// TwinCAT 3 PLC project PLC_PROJ
// ProgramVersion: 3.1.4026.15
// libraries:
//   Tc2_EtherCAT, * (Beckhoff Automation GmbH)
//   Tc2_IoFunctions, * (Beckhoff Automation GmbH)
//   Tc2_SerialCom, * (Beckhoff Automation GmbH)
//   Tc2_Standard, * (Beckhoff Automation GmbH)
//   Tc2_System, * (Beckhoff Automation GmbH)
// project tree:
//   DUTs/ CAN_IFACE_QUEUE.TcDUT, CAN_MSG.TcDUT, CAN_MsgSlot.TcDUT
//   GVLs/ ANALOG.TcGVL, EL6751_GVLs.TcGVL, GLOBAL_VARS.TcGVL
//   / PlcTask.TcTTO
//   POUs/CanHelpers/ F_ComposeSlot.TcPOU, F_ParseSlot.TcPOU
//   POUs/ MAIN.TcPOU
//   POUs/PsuHelpers/ BytesToUInt16.TcPOU, CurrentToRaw.TcPOU, RawToCurrent.TcPOU, RawToVoltage.TcPOU, VoltageToRaw.TcPOU
//   POUs/PsuIface/ FB_PowerSupply.TcPOU
// real-time tasks:
//   TASK PlcTask: cycle T#100000us, priority 20, ADS port 350
// I/O:
//   DEVICE Device 1 (EtherCAT), AmsNetId 5.156.240.208.2.1
//     Term 1 (EK1200) [EK1200-7000 EtherCAT Power supply (1,5A E-Bus)]
//       Term 2 (EL2008) [EL2008 8Ch. Dig. Output 24V, 0.5A]
//       Term 3 (EL3174-0042) [EL3174-0042 4Ch. Ana. Input +/-30V, +/-60V 16 Bit, Isolated Channels]
//       Term 4 (EL3692) [EL3692 2Ch. resistance measurement terminal]
//       Term 5 (EL6751) [EL6751 CANopen Master]
//       Term 6 (EL6631) [EL6631 PROFINET IO Controller]
//       Term 7 (EL9011) [EL9011 End Terminal]
//   DEVICE Device 2 (NOV-DP-RAM)
//   DEVICE Device 3 (Onboard I/O Device), AmsNetId 5.156.240.208.4.1
//     Term 1 (CX7028) [CX7028-0000-0121]
//       modules: Module 1 (DIO_2x), Module 2 (Empty Module), Module 3 (DIO_2x), Module 4 (Empty Module), Module 5 (DI_2x), Module 6 (Empty Module), Module 7 (DI_2x), Module 8 (Empty Module)
//   DEVICE Device 4 (COM Port)
//   DEVICE Device 5 (COM Port)
//   DEVICE Device 6 (EL6751), AmsNetId 5.156.240.208.7.1
//     Box 9 (CAN Interface)
// variable links:
//   PLC_PROJ/PLC_PROJ Instance <-> Device 1 (EtherCAT)/Term 1 (EK1200)/Term 2 (EL2008)
//     PlcTask Outputs/GLOBAL_VARS.DO_EL2008_OUT_2 <-> Channel 2/Output
//     PlcTask Outputs/GLOBAL_VARS.DO_EL2008_OUT_4 <-> Channel 4/Output
//     PlcTask Outputs/GLOBAL_VARS.DO_EL2008_OUT_5 <-> Channel 5/Output
//     PlcTask Outputs/GLOBAL_VARS.DO_EL2008_OUT_6 <-> Channel 6/Output
//     PlcTask Outputs/GLOBAL_VARS.DO_EL2008_OUT_7 <-> Channel 7/Output
//     PlcTask Outputs/GLOBAL_VARS.DO_EL2008_OUT_8 <-> Channel 8/Output
//     PlcTask Outputs/GLOBAL_VARS.DO_EL2008_RELAY_0 <-> Channel 1/Output
//     PlcTask Outputs/GLOBAL_VARS.DO_EL2008_RELAY_1 <-> Channel 3/Output
//   PLC_PROJ/PLC_PROJ Instance <-> Device 4 (COM Port)
//     PlcTask Inputs/GLOBAL_VARS.X003_In/D[0] <-> Inputs/Data1
//     PlcTask Inputs/GLOBAL_VARS.X003_In/D[10] <-> Inputs/Data11
//     PlcTask Inputs/GLOBAL_VARS.X003_In/D[11] <-> Inputs/Data12
//     PlcTask Inputs/GLOBAL_VARS.X003_In/D[12] <-> Inputs/Data13
//     PlcTask Inputs/GLOBAL_VARS.X003_In/D[13] <-> Inputs/Data14
//     PlcTask Inputs/GLOBAL_VARS.X003_In/D[14] <-> Inputs/Data15
//     PlcTask Inputs/GLOBAL_VARS.X003_In/D[15] <-> Inputs/Data16
//     PlcTask Inputs/GLOBAL_VARS.X003_In/D[16] <-> Inputs/Data17
//     PlcTask Inputs/GLOBAL_VARS.X003_In/D[17] <-> Inputs/Data18
//     PlcTask Inputs/GLOBAL_VARS.X003_In/D[18] <-> Inputs/Data19
//     PlcTask Inputs/GLOBAL_VARS.X003_In/D[19] <-> Inputs/Data20
//     PlcTask Inputs/GLOBAL_VARS.X003_In/D[1] <-> Inputs/Data2
//     PlcTask Inputs/GLOBAL_VARS.X003_In/D[20] <-> Inputs/Data21
//     PlcTask Inputs/GLOBAL_VARS.X003_In/D[21] <-> Inputs/Data22
//     PlcTask Inputs/GLOBAL_VARS.X003_In/D[22] <-> Inputs/Data23
//     PlcTask Inputs/GLOBAL_VARS.X003_In/D[23] <-> Inputs/Data24
//     PlcTask Inputs/GLOBAL_VARS.X003_In/D[24] <-> Inputs/Data25
//     PlcTask Inputs/GLOBAL_VARS.X003_In/D[25] <-> Inputs/Data26
//     PlcTask Inputs/GLOBAL_VARS.X003_In/D[26] <-> Inputs/Data27
//     PlcTask Inputs/GLOBAL_VARS.X003_In/D[27] <-> Inputs/Data28
//     PlcTask Inputs/GLOBAL_VARS.X003_In/D[28] <-> Inputs/Data29
//     PlcTask Inputs/GLOBAL_VARS.X003_In/D[29] <-> Inputs/Data30
//     PlcTask Inputs/GLOBAL_VARS.X003_In/D[2] <-> Inputs/Data3
//     PlcTask Inputs/GLOBAL_VARS.X003_In/D[30] <-> Inputs/Data31
//     PlcTask Inputs/GLOBAL_VARS.X003_In/D[31] <-> Inputs/Data32
//     PlcTask Inputs/GLOBAL_VARS.X003_In/D[32] <-> Inputs/Data33
//     PlcTask Inputs/GLOBAL_VARS.X003_In/D[33] <-> Inputs/Data34
//     PlcTask Inputs/GLOBAL_VARS.X003_In/D[34] <-> Inputs/Data35
//     PlcTask Inputs/GLOBAL_VARS.X003_In/D[35] <-> Inputs/Data36
//     PlcTask Inputs/GLOBAL_VARS.X003_In/D[36] <-> Inputs/Data37
//     PlcTask Inputs/GLOBAL_VARS.X003_In/D[37] <-> Inputs/Data38
//     PlcTask Inputs/GLOBAL_VARS.X003_In/D[38] <-> Inputs/Data39
//     PlcTask Inputs/GLOBAL_VARS.X003_In/D[39] <-> Inputs/Data40
//     PlcTask Inputs/GLOBAL_VARS.X003_In/D[3] <-> Inputs/Data4
//     PlcTask Inputs/GLOBAL_VARS.X003_In/D[40] <-> Inputs/Data41
//     PlcTask Inputs/GLOBAL_VARS.X003_In/D[41] <-> Inputs/Data42
//     PlcTask Inputs/GLOBAL_VARS.X003_In/D[42] <-> Inputs/Data43
//     PlcTask Inputs/GLOBAL_VARS.X003_In/D[43] <-> Inputs/Data44
//     PlcTask Inputs/GLOBAL_VARS.X003_In/D[44] <-> Inputs/Data45
//     PlcTask Inputs/GLOBAL_VARS.X003_In/D[45] <-> Inputs/Data46
//     PlcTask Inputs/GLOBAL_VARS.X003_In/D[46] <-> Inputs/Data47
//     PlcTask Inputs/GLOBAL_VARS.X003_In/D[47] <-> Inputs/Data48
//     PlcTask Inputs/GLOBAL_VARS.X003_In/D[48] <-> Inputs/Data49
//     PlcTask Inputs/GLOBAL_VARS.X003_In/D[49] <-> Inputs/Data50
//     PlcTask Inputs/GLOBAL_VARS.X003_In/D[4] <-> Inputs/Data5
//     PlcTask Inputs/GLOBAL_VARS.X003_In/D[50] <-> Inputs/Data51
//     PlcTask Inputs/GLOBAL_VARS.X003_In/D[51] <-> Inputs/Data52
//     PlcTask Inputs/GLOBAL_VARS.X003_In/D[52] <-> Inputs/Data53
//     PlcTask Inputs/GLOBAL_VARS.X003_In/D[53] <-> Inputs/Data54
//     PlcTask Inputs/GLOBAL_VARS.X003_In/D[54] <-> Inputs/Data55
//     PlcTask Inputs/GLOBAL_VARS.X003_In/D[55] <-> Inputs/Data56
//     PlcTask Inputs/GLOBAL_VARS.X003_In/D[56] <-> Inputs/Data57
//     PlcTask Inputs/GLOBAL_VARS.X003_In/D[57] <-> Inputs/Data58
//     PlcTask Inputs/GLOBAL_VARS.X003_In/D[58] <-> Inputs/Data59
//     PlcTask Inputs/GLOBAL_VARS.X003_In/D[59] <-> Inputs/Data60
//     PlcTask Inputs/GLOBAL_VARS.X003_In/D[5] <-> Inputs/Data6
//     PlcTask Inputs/GLOBAL_VARS.X003_In/D[60] <-> Inputs/Data61
//     PlcTask Inputs/GLOBAL_VARS.X003_In/D[61] <-> Inputs/Data62
//     PlcTask Inputs/GLOBAL_VARS.X003_In/D[62] <-> Inputs/Data63
//     PlcTask Inputs/GLOBAL_VARS.X003_In/D[63] <-> Inputs/Data64
//     PlcTask Inputs/GLOBAL_VARS.X003_In/D[6] <-> Inputs/Data7
//     PlcTask Inputs/GLOBAL_VARS.X003_In/D[7] <-> Inputs/Data8
//     PlcTask Inputs/GLOBAL_VARS.X003_In/D[8] <-> Inputs/Data9
//     PlcTask Inputs/GLOBAL_VARS.X003_In/D[9] <-> Inputs/Data10
//     PlcTask Inputs/GLOBAL_VARS.X003_In/SerStatus <-> Inputs/Status
//     PlcTask Outputs/GLOBAL_VARS.X003_Out/D[0] <-> Outputs/Data1
//     PlcTask Outputs/GLOBAL_VARS.X003_Out/D[10] <-> Outputs/Data11
//     PlcTask Outputs/GLOBAL_VARS.X003_Out/D[11] <-> Outputs/Data12
//     PlcTask Outputs/GLOBAL_VARS.X003_Out/D[12] <-> Outputs/Data13
//     PlcTask Outputs/GLOBAL_VARS.X003_Out/D[13] <-> Outputs/Data14
//     PlcTask Outputs/GLOBAL_VARS.X003_Out/D[14] <-> Outputs/Data15
//     PlcTask Outputs/GLOBAL_VARS.X003_Out/D[15] <-> Outputs/Data16
//     PlcTask Outputs/GLOBAL_VARS.X003_Out/D[16] <-> Outputs/Data17
//     PlcTask Outputs/GLOBAL_VARS.X003_Out/D[17] <-> Outputs/Data18
//     PlcTask Outputs/GLOBAL_VARS.X003_Out/D[18] <-> Outputs/Data19
//     PlcTask Outputs/GLOBAL_VARS.X003_Out/D[19] <-> Outputs/Data20
//     PlcTask Outputs/GLOBAL_VARS.X003_Out/D[1] <-> Outputs/Data2
//     PlcTask Outputs/GLOBAL_VARS.X003_Out/D[20] <-> Outputs/Data21
//     PlcTask Outputs/GLOBAL_VARS.X003_Out/D[21] <-> Outputs/Data22
//     PlcTask Outputs/GLOBAL_VARS.X003_Out/D[22] <-> Outputs/Data23
//     PlcTask Outputs/GLOBAL_VARS.X003_Out/D[23] <-> Outputs/Data24
//     PlcTask Outputs/GLOBAL_VARS.X003_Out/D[24] <-> Outputs/Data25
//     PlcTask Outputs/GLOBAL_VARS.X003_Out/D[25] <-> Outputs/Data26
//     PlcTask Outputs/GLOBAL_VARS.X003_Out/D[26] <-> Outputs/Data27
//     PlcTask Outputs/GLOBAL_VARS.X003_Out/D[27] <-> Outputs/Data28
//     PlcTask Outputs/GLOBAL_VARS.X003_Out/D[28] <-> Outputs/Data29
//     PlcTask Outputs/GLOBAL_VARS.X003_Out/D[29] <-> Outputs/Data30
//     PlcTask Outputs/GLOBAL_VARS.X003_Out/D[2] <-> Outputs/Data3
//     PlcTask Outputs/GLOBAL_VARS.X003_Out/D[30] <-> Outputs/Data31
//     PlcTask Outputs/GLOBAL_VARS.X003_Out/D[31] <-> Outputs/Data32
//     PlcTask Outputs/GLOBAL_VARS.X003_Out/D[32] <-> Outputs/Data33
//     PlcTask Outputs/GLOBAL_VARS.X003_Out/D[33] <-> Outputs/Data34
//     PlcTask Outputs/GLOBAL_VARS.X003_Out/D[34] <-> Outputs/Data35
//     PlcTask Outputs/GLOBAL_VARS.X003_Out/D[35] <-> Outputs/Data36
//     PlcTask Outputs/GLOBAL_VARS.X003_Out/D[36] <-> Outputs/Data37
//     PlcTask Outputs/GLOBAL_VARS.X003_Out/D[37] <-> Outputs/Data38
//     PlcTask Outputs/GLOBAL_VARS.X003_Out/D[38] <-> Outputs/Data39
//     PlcTask Outputs/GLOBAL_VARS.X003_Out/D[39] <-> Outputs/Data40
//     PlcTask Outputs/GLOBAL_VARS.X003_Out/D[3] <-> Outputs/Data4
//     PlcTask Outputs/GLOBAL_VARS.X003_Out/D[40] <-> Outputs/Data41
//     PlcTask Outputs/GLOBAL_VARS.X003_Out/D[41] <-> Outputs/Data42
//     PlcTask Outputs/GLOBAL_VARS.X003_Out/D[42] <-> Outputs/Data43
//     PlcTask Outputs/GLOBAL_VARS.X003_Out/D[43] <-> Outputs/Data44
//     PlcTask Outputs/GLOBAL_VARS.X003_Out/D[44] <-> Outputs/Data45
//     PlcTask Outputs/GLOBAL_VARS.X003_Out/D[45] <-> Outputs/Data46
//     PlcTask Outputs/GLOBAL_VARS.X003_Out/D[46] <-> Outputs/Data47
//     PlcTask Outputs/GLOBAL_VARS.X003_Out/D[47] <-> Outputs/Data48
//     PlcTask Outputs/GLOBAL_VARS.X003_Out/D[48] <-> Outputs/Data49
//     PlcTask Outputs/GLOBAL_VARS.X003_Out/D[49] <-> Outputs/Data50
//     PlcTask Outputs/GLOBAL_VARS.X003_Out/D[4] <-> Outputs/Data5
//     PlcTask Outputs/GLOBAL_VARS.X003_Out/D[50] <-> Outputs/Data51
//     PlcTask Outputs/GLOBAL_VARS.X003_Out/D[51] <-> Outputs/Data52
//     PlcTask Outputs/GLOBAL_VARS.X003_Out/D[52] <-> Outputs/Data53
//     PlcTask Outputs/GLOBAL_VARS.X003_Out/D[53] <-> Outputs/Data54
//     PlcTask Outputs/GLOBAL_VARS.X003_Out/D[54] <-> Outputs/Data55
//     PlcTask Outputs/GLOBAL_VARS.X003_Out/D[55] <-> Outputs/Data56
//     PlcTask Outputs/GLOBAL_VARS.X003_Out/D[56] <-> Outputs/Data57
//     PlcTask Outputs/GLOBAL_VARS.X003_Out/D[57] <-> Outputs/Data58
//     PlcTask Outputs/GLOBAL_VARS.X003_Out/D[58] <-> Outputs/Data59
//     PlcTask Outputs/GLOBAL_VARS.X003_Out/D[59] <-> Outputs/Data60
//     PlcTask Outputs/GLOBAL_VARS.X003_Out/D[5] <-> Outputs/Data6
//     PlcTask Outputs/GLOBAL_VARS.X003_Out/D[60] <-> Outputs/Data61
//     PlcTask Outputs/GLOBAL_VARS.X003_Out/D[61] <-> Outputs/Data62
//     PlcTask Outputs/GLOBAL_VARS.X003_Out/D[62] <-> Outputs/Data63
//     PlcTask Outputs/GLOBAL_VARS.X003_Out/D[63] <-> Outputs/Data64
//     PlcTask Outputs/GLOBAL_VARS.X003_Out/D[6] <-> Outputs/Data7
//     PlcTask Outputs/GLOBAL_VARS.X003_Out/D[7] <-> Outputs/Data8
//     PlcTask Outputs/GLOBAL_VARS.X003_Out/D[8] <-> Outputs/Data9
//     PlcTask Outputs/GLOBAL_VARS.X003_Out/D[9] <-> Outputs/Data10
//     PlcTask Outputs/GLOBAL_VARS.X003_Out/SerCtrl <-> Outputs/Ctrl
//   PLC_PROJ/PLC_PROJ Instance <-> Device 6 (EL6751)/Box 9 (CAN Interface)
//     PlcTask Inputs/EL6751_GVLs.gCanIf_RxMsg <-> Inputs/RxQueue
//     PlcTask Outputs/EL6751_GVLs.gCanIf_TxMsg <-> Outputs/TxQueue

CONFIGURATION PLC_PROJ
    RESOURCE PLC ON TwinCAT3
        TASK PlcTask(INTERVAL := T#100000us, PRIORITY := 20);
        PROGRAM MAIN WITH PlcTask : MAIN;
    END_RESOURCE
END_CONFIGURATION

// ---- DUTs/CAN_IFACE_QUEUE.TcDUT
TYPE CAN_IFACE_QUEUE :
STRUCT
	TxCounter      : UINT;
	RxCounter      : UINT;
	NoOfMessages : UINT;
	Messages     : ARRAY[0..9] OF CAN_MsgSlot; 
END_STRUCT
END_TYPE

// ---- DUTs/CAN_MSG.TcDUT
TYPE CAN_MSG :
STRUCT
	ID   : UDINT; // Unsigned 32-bit
	DLC  : BYTE;  // Unsigned 8-bit
	DATA : ARRAY[0..7] OF BYTE;
END_STRUCT
END_TYPE

// ---- DUTs/CAN_MsgSlot.TcDUT
TYPE CAN_MsgSlot :
STRUCT
	cobId : UINT; // Unsigned 16-bit
    data  : ARRAY[0..7] OF BYTE;
END_STRUCT
END_TYPE

// ---- GVLs/ANALOG.TcGVL

{attribute 'qualified_only'}
VAR_GLOBAL
	AL_1 AT %I* : INT;
	AL_2 AT %I* : INT;
	AL_3 AT %I* : INT;
	AL_4 AT %I* : INT;
END_VAR

// ---- GVLs/EL6751_GVLs.TcGVL
{attribute 'qualified_only'}
VAR_GLOBAL
	gCanIf_TxMsg         AT %Q* : CAN_IFACE_QUEUE;
	gCanIf_RxMsg         AT %I* : CAN_IFACE_QUEUE;
END_VAR

// ---- GVLs/GLOBAL_VARS.TcGVL
(* GVLs/GLOBAL_VARS *)

{attribute 'qualified_only'}
VAR_GLOBAL
    DO_EL2008_RELAY_0    AT %Q* : BOOL;   // EL2008 channel 1
    DO_EL2008_RELAY_1    AT %Q* : BOOL;   // EL2008 channel 3
	DO_EL2008_OUT_2      AT %Q* : BOOL;   // EL2008 channel 2
	DO_EL2008_OUT_4      AT %Q* : BOOL;   // EL2008 channel 4
	DO_EL2008_OUT_5      AT %Q* : BOOL;   // EL2008 channel 5
	DO_EL2008_OUT_6      AT %Q* : BOOL;   // EL2008 channel 6
	DO_EL2008_OUT_7      AT %Q* : BOOL;   // EL2008 channel 7
	DO_EL2008_OUT_8      AT %Q* : BOOL;   // EL2008 channel 8

  	X003_Out             AT %Q* : PcComOutData;
  	X003_In              AT %I* : PcComInData;
END_VAR

// ---- POUs/MAIN.TcPOU
(* POUs/MAIN *)

PROGRAM MAIN
VAR
	CanRx          : CAN_IFACE_QUEUE;
	CanTx          : CAN_IFACE_QUEUE;
	i              : UINT;
	relayIdx       : UINT;
	slotIn         : CAN_MsgSlot;
	slotOut        : CAN_MsgSlot;
	msgIn          : CAN_MSG;
	msgOut         : CAN_MSG;

	rawVoltIn      : UINT := 0;
	rawVoltOut     : UINT := 0;
	rawCurrentIn   : UINT := 0;
	rawCurrentOut  : UINT := 0;

	physVoltIn     : REAL := 0.0;
	physVoltOut    : REAL := 0.0;
	physCurrentIn  : REAL := 0.0;
	physCurrentOut : REAL := 0.0;

	FB_PSU         : FB_PowerSupply;
	
	feedbackTmr    : TON;    // On-delay timer for periodic feedback
	feedbackReq    : BOOL;   // Pulses TRUE once every 100 ms when Q rises

	ALGO_RUN       : BOOL := FALSE;
END_VAR


FB_PSU.Cycle();



IF ALGO_RUN THEN

	feedbackTmr(IN := TRUE, PT := T#100MS);  
	feedbackReq := feedbackTmr.Q;  
	IF feedbackReq THEN  
	  feedbackTmr(IN := FALSE);  
	END_IF  

	// When timer fires, send voltage and current feedback
	IF feedbackReq THEN

		GLOBAL_VARS.DO_EL2008_RELAY_0 := ANALOG.AL_2 <= 20000;
		GLOBAL_VARS.DO_EL2008_RELAY_1 := ANALOG.AL_2 > 20000;

		// Read latest physical values
		physVoltIn := FB_PSU.GetVoltage();
		rawVoltIn := VoltageToRaw(volts := physVoltIn);
		physCurrentIn := FB_PSU.GetCurrent();
		rawCurrentIn := CurrentToRaw(amps := physCurrentIn);

		// Read back voltage and compose 0x201
		msgOut.ID  := 16#201;
		msgOut.DLC := 2;
		msgOut.DATA[1] := TO_BYTE(SHR(rawVoltIn, 8));   // MSB
		msgOut.DATA[0] := TO_BYTE(rawVoltIn AND 16#FF); // LSB
		slotOut := F_ComposeSlot(msg := msgOut);
		CanTx.Messages[0] := slotOut;

		// Read back current and compose 0x301
		msgOut.ID  := 16#301;
		msgOut.DLC := 2;
		msgOut.DATA[1] := TO_BYTE(SHR(rawCurrentIn, 8));
		msgOut.DATA[0] := TO_BYTE(rawCurrentIn AND 16#FF);
		slotOut := F_ComposeSlot(msg := msgOut);
		CanTx.Messages[1] := slotOut;

		// Finalize and trigger EtherCAT send
		CanTx.NoOfMessages := 2;
		CanTx.TxCounter    := EL6751_GVLs.gCanIf_TxMsg.TxCounter + 1;
		EL6751_GVLs.gCanIf_TxMsg := CanTx;
	END_IF


	CanRx := EL6751_GVLs.gCanIf_RxMsg; // Create a copy of the hardware mapped CAN Rx Queue
	// Process all received messages
	IF CanRx.NoOfMessages > 0 THEN
		FOR i := 0 TO CanRx.NoOfMessages - 1 DO
			slotIn := CanRx.Messages[i];
			msgIn := F_ParseSlot(slot := slotIn);
	
			// Handle by CAN ID
			CASE msgIn.ID OF
	
			16#100:  // Relay control
				IF msgIn.DLC = 8 THEN
					// GLOBAL_VARS.DO_EL2008_RELAY_0 := msgIn.DATA[0] = 1;
					// GLOBAL_VARS.DO_EL2008_RELAY_1 := msgIn.DATA[1] = 1;
				END_IF;

			16#200:  // Voltage control
				IF msgIn.DLC = 2 THEN
					rawVoltOut := BytesToUInt16(highByte := msgIn.DATA[1], lowByte := msgIn.DATA[0]);
					physVoltOut := RawToVoltage(raw := rawVoltOut);
					FB_PSU.SetVoltage(volts := physVoltOut);
				END_IF;

			16#300:  // Current control
				IF msgIn.DLC = 2 THEN
					rawCurrentOut := SHL(TO_UINT(msgIn.DATA[1]), 8) OR TO_UINT(msgIn.DATA[0]);
					physCurrentOut := RawToCurrent(raw := rawCurrentOut);
					FB_PSU.SetCurrent(amps := physCurrentOut);
				END_IF;

			END_CASE;
		END_FOR
	END_IF
END_IF

END_PROGRAM

// ---- POUs/PsuIface/FB_PowerSupply.TcPOU
FUNCTION_BLOCK FB_PowerSupply
VAR
	pComIn     : POINTER TO BYTE;
	SizeComIn  : UDINT;
	pComOut    : POINTER TO BYTE;
	SizeComOut : UDINT;

	fbPort   : SerialLineControl;  // call every scan
	fbSend   : SendString;
	fbRecv   : ReceiveString;
	fbClearRx : ClearComBuffer;

	_bufTx   : ComBuffer;          // your existing TxBuf
	_bufRx   : ComBuffer;          // your existing RxBuf

	_txErr   : ComError_t;
	_rxErr   : ComError_t;
	_txBusy  : BOOL;
	_rxBusy  : BOOL;
	_Vrecvd  : BOOL;
	_Irecvd  : BOOL;

	trigRecvReset : R_TRIG;
	
	lastVoltage : REAL;
	lastCurrent : REAL;

END_VAR

METHOD Cycle
IF NOT fbPort.initialized THEN
  	_bufTx.RdIdx    := 0;
	_bufTx.WrIdx    := 0;
	_bufTx.Count    := 0;
	_bufTx.FreeByte := SIZEOF(_bufTx.Buffer);
	_bufTx.Error    := 0;
	_bufTx.blocked  := FALSE;

	_bufRx.RdIdx    := 0;
	_bufRx.WrIdx    := 0;
	_bufRx.Count    := 0;
	_bufRx.FreeByte := SIZEOF(_bufRx.Buffer);
	_bufRx.Error    := 0;
	_bufRx.blocked  := FALSE;
END_IF

fbPort(
    Mode      := SERIALLINEMODE_DEFAULT,
    pComIn    := ADR(GLOBAL_VARS.X003_In),
    pComOut   := ADR(GLOBAL_VARS.X003_Out),
    SizeComIn := SIZEOF(GLOBAL_VARS.X003_In),
    TxBuffer  := _bufTx,
    RxBuffer  := _bufRx
);
END_METHOD

METHOD GetCurrent : REAL

VAR
	temp_str : STRING(80);
END_VAR
Cycle();

// 1) Send the command
fbSend(
	SendString := CONCAT('ISET1?', CHR(10)),
	TxBuffer   := _bufTx,
	Busy       => _txBusy
);

// 2) Detect the instant that Busy goes TRUE → FALSE
trigRecvReset(CLK := _txBusy);

Cycle();

// 3) Call fbRecv _every_ scan, but only reset it on that one‐scan pulse
fbRecv(
	Reset          := trigRecvReset.Q,  // TRUE _only_ the scan after sendDone
	Suffix         := CHR(10),
	Timeout        := T#0ms,
	RxBuffer       := _bufRx,
	ReceivedString := temp_str,
	StringReceived => _Irecvd,
	busy           => ,
	Error          => _rxErr
);

// only update when a fresh line arrived without error
IF (_rxErr = COMERROR_NOERROR) AND _Irecvd THEN
    lastCurrent := STRING_TO_REAL(temp_str);
END_IF

// always return the last known good value
GetCurrent := lastCurrent;
END_METHOD

METHOD GetVoltage : REAL

VAR
	temp_str : STRING(80);
END_VAR
Cycle();

// 1) Send the command
fbSend(
	SendString := CONCAT('VSET1?', CHR(10)),
	TxBuffer   := _bufTx,
	Busy       => _txBusy
);

// 2) Detect the instant that Busy goes TRUE → FALSE
trigRecvReset(CLK := _txBusy);

Cycle();

// 3) Call fbRecv _every_ scan, but only reset it on that one‐scan pulse
fbRecv(
	Reset          := trigRecvReset.Q,  // TRUE _only_ the scan after sendDone
	Suffix         := CHR(10),
	Timeout        := T#0ms,
	RxBuffer       := _bufRx,
	ReceivedString := temp_str,
	StringReceived => _Vrecvd,
	busy           => ,
	Error          => _rxErr
);

// only update when a fresh line arrived without error
IF (_rxErr = COMERROR_NOERROR) AND _Vrecvd THEN
    lastVoltage := STRING_TO_REAL(temp_str);
	fbClearRx(Buffer := _bufRx);
END_IF

// always return the last known good value
GetVoltage := lastVoltage;
END_METHOD

METHOD SetCurrent

VAR_INPUT
	amps : REAL;
END_VAR

VAR
	raw    : UINT;
	hiPart : UINT;
	loPart : UINT;  
  	loStr  : STRING(3);
	hiStr  : STRING(3);
	txStr  : STRING(20);
END_VAR
Cycle();

raw := VoltageToRaw(amps);

// build “VSET1:xx.yy”  
hiPart := raw / 100;         // integral volts
loPart := raw MOD 100;       // thousandts
loStr  := UINT_TO_STRING(loPart);

IF loPart < 10 THEN  
	loStr := CONCAT('0', loStr);  
END_IF;  
hiStr  := UINT_TO_STRING(hiPart);  

txStr := CONCAT(CONCAT('ISET1:', CONCAT(hiStr, CONCAT('.', loStr))), CHR(10));  

fbSend(
	SendString := txStr,
	TxBuffer   := _bufTx,
	Error      => _txErr
);
END_METHOD

METHOD SetVoltage

VAR_INPUT
	volts : REAL;
END_VAR

VAR
	raw    : UINT;
	hiPart : UINT;
	loPart : UINT;  
  	loStr  : STRING(3);
	hiStr  : STRING(3);
	txStr  : STRING(20);
END_VAR
Cycle();

raw := VoltageToRaw(volts);

// build “VSET1:xx.yy”  
hiPart := raw / 100;         // integral volts  
loPart := raw MOD 100;       // hundredths  
loStr  := UINT_TO_STRING(loPart);  
IF loPart < 10 THEN  
	loStr := CONCAT('0', loStr);  
END_IF;  
hiStr  := UINT_TO_STRING(hiPart);  

txStr := CONCAT(CONCAT('VSET1:', CONCAT(hiStr, CONCAT('.', loStr))), CHR(10));  

fbSend(
	SendString := txStr,
	TxBuffer   := _bufTx,
	Error      => _txErr
);
END_METHOD

END_FUNCTION_BLOCK

// ---- POUs/PsuHelpers/VoltageToRaw.TcPOU
FUNCTION VoltageToRaw : UINT
VAR_INPUT
	volts : REAL;          // 0.00 to 60.00
END_VAR
VAR
  tmp : REAL;
END_VAR


tmp := volts * 100.0;

IF tmp < 0.0 THEN
	tmp := 0.0;
ELSIF tmp > 6000.0 THEN
	tmp := 6000.0;
END_IF

VoltageToRaw := REAL_TO_UINT(tmp);

END_FUNCTION

// ---- POUs/PsuHelpers/CurrentToRaw.TcPOU
FUNCTION CurrentToRaw : UINT

VAR_INPUT
  amps : REAL;           // 0.00 to 5.00
END_VAR

VAR
  tmp : REAL; // 0 to 5000
END_VAR


tmp := amps * 1000.0;

IF tmp < 0.0 THEN
	tmp := 0.0;
ELSIF tmp > 5000.0 THEN
	tmp := 5000.0;
END_IF;

CurrentToRaw := REAL_TO_UINT(tmp);

END_FUNCTION

// ---- POUs/CanHelpers/F_ComposeSlot.TcPOU
FUNCTION F_ComposeSlot : CAN_MsgSlot

VAR_INPUT
    msg : CAN_MSG;        // your prepared CAN message
END_VAR

VAR
    packedID : UINT;
    i        : INT;
END_VAR

// 1) Pack ID into bits 5..15, ensure it’s ≤ 0x07FF
packedID := SHL(TO_UINT(msg.ID AND 16#07FF), 5);

// 2) OR in the DLC (lower nibble), ensure it’s ≤ 8
packedID := packedID OR (TO_UINT(msg.DLC AND 16#000F));

// 3) Fill result
F_ComposeSlot.cobId := packedID;

// 4) Copy data bytes
FOR i := 0 TO TO_INT(msg.DLC) - 1 DO
    F_ComposeSlot.data[i] := msg.DATA[i];
END_FOR

// Zero out any unused bytes (optional)
FOR i := TO_INT(msg.DLC) TO 7 DO
    F_ComposeSlot.data[i] := 0;
END_FOR

END_FUNCTION

// ---- POUs/CanHelpers/F_ParseSlot.TcPOU
FUNCTION F_ParseSlot : CAN_MSG

VAR_INPUT
	slot : CAN_MsgSlot;    // the raw slot from EL6751
END_VAR

VAR
    tmpID  : UINT;
    tmpDLC : UINT;
    i      : INT;
END_VAR

// 1) Extract the 11-bit ID
tmpID := SHR(slot.cobId, 5);           // bits 5..15

// 2) Extract the 4-bit DLC
tmpDLC := slot.cobId AND 16#000F;      // bits 0..3

// 3) Fill result
F_ParseSlot.ID  := tmpID;             // widens UINT → UDINT
F_ParseSlot.DLC := TO_BYTE(tmpDLC);

// 4) Copy up to 8 data bytes
FOR i := 0 TO TO_INT(F_ParseSlot.DLC) - 1 DO
    F_ParseSlot.DATA[i] := slot.data[i];
END_FOR

// Zero out any unused bytes (optional)
FOR i := TO_INT(F_ParseSlot.DLC) TO 7 DO
    F_ParseSlot.DATA[i] := 0;
END_FOR

END_FUNCTION

// ---- POUs/PsuHelpers/BytesToUInt16.TcPOU
FUNCTION BytesToUInt16 : UINT

VAR_INPUT
  highByte : BYTE;  // Most‐significant byte
  lowByte  : BYTE;  // Least‐significant byte
END_VAR

VAR
  _hb  : UINT;
  _lb  : UINT;
END_VAR


// Shift the high byte into bits 8–15, then OR in the low byte
_hb := SHL( TO_UINT(highByte), 8 );
_lb := TO_UINT(lowByte);
BytesToUInt16 := _hb OR _lb;

END_FUNCTION

// ---- POUs/PsuHelpers/RawToVoltage.TcPOU
FUNCTION RawToVoltage : REAL
VAR_INPUT
	raw : UINT;            // 0 to 6000
END_VAR


RawToVoltage := UINT_TO_REAL(raw) * 0.01;  // 0.00 to 60.00 V

END_FUNCTION

// ---- POUs/PsuHelpers/RawToCurrent.TcPOU
FUNCTION RawToCurrent : REAL
VAR_INPUT
	raw : UINT;            // 0 to 5000
END_VAR


RawToCurrent := UINT_TO_REAL(raw) * 0.001;  // → 0.00 to 5.00 A

END_FUNCTION
